{attribute 'qualified_only'}
{attribute 'strict'}
TYPE SystemStatus :
(
	System_OK := 0,
	ChassisManual_Slow,
	ChassisManual_Fast,
	EmergencyStop:=255
);
END_TYPE

(* stored: Version 1.1.0.1, ProductVersion 3.1.4024.14
   DUT SystemStatus: Id {8ac778b6-2158-46dc-ac60-814e8fd39e9b} *)
